{attribute addProperty BoxType "EL3681-0000-0017"}
{attribute addProperty Id "SettingAT %I*Setting_7AA6B313162"}
{attribute addProperty CRC "3207721882"}
{attribute addProperty SizeInBites "16"}
{attribute addProperty SizeInBytes "2"}
TYPE SAI_Range_BF31F39A :
STRUCT
	{attribute addProperty Name "Setting"}
	Setting AT %I* : Setting_7AA6B313;
END_STRUCT
END_TYPE

(* stored: Version 1.2.0.0, ProductVersion 3.1.4024.9
   DUT SAI_Range_BF31F39A: Id {94dd4a45-fd3d-4338-9f59-7c9acb985d4e} *)
